(* PLC project 117_1_V0.5.project, CODESYS CODESYS V3.5 SP17 Patch 3 *)
(* stored: creationDateTime 1970-01-01T00:00:00, modificationDateTime 2026-03-26T18:14:32.4070562 *)

{attribute 'strict'}
TYPE ALL_DI : (inLiveCircuitsDC, inFirstAlarmMushroom, inSecondAlarmMushroom, inLiveCircuitsAC, inUpsDC_OK, inUpsBattaryBad, inUpsBattaryWork, inUpperLimitSwitch, inLowerLimitSwitch, inRemovingLimitSwitch, inExciter, inBit11, inBit12, inLeftDoor, inRightDoor, inBit15);
END_TYPE
